Fanuc TP program (LS listing): CLOSE_CHUCK_2.LS

/PROG  CLOSE_CHUCK_2
/ATTR
OWNER		= MNEDITOR;
COMMENT		= "";
PROG_SIZE	= 146;
CREATE		= DATE 19-01-28  TIME 18:39:14;
MODIFIED	= DATE 21-01-31  TIME 12:33:18;
FILE_NAME	= ;
VERSION		= 0;
LINE_COUNT	= 1;
MEMORY_SIZE	= 514;
PROTECT		= READ_WRITE;
TCD:  STACK_SIZE	= 0,
      TASK_PRIORITY	= 50,
      TIME_SLICE	= 0,
      BUSY_LAMP_OFF	= 0,
      ABORT_REQUEST	= 0,
      PAUSE_REQUEST	= 0;
DEFAULT_GROUP	= 1,*,*,*,*;
CONTROL_CODE	= 00000000 00000000;
/APPL
/MN
   1:  RO[2]=OFF ;
/POS
/END
